(* IEC 61131-3 sources: teller/JD_Teller_LC2_V11/Class/_AlarmX0Para, 1 file *)

(* ---- _AlarmX0Para.st ---- *)
(*!
<Class
	Name               = "_AlarmX0Para"
	Revision           = "0.4"
	RealtimeTask       = "false"
	CyclicTask         = "false"
	BackgroundTask     = "false"
	Sigmatek           = "true"
	OSInterface        = "false"
	HighPriority       = "false"
	Automatic          = "false"
	UpdateMode         = "Prescan"
	SharedCommandTable = "true"
	Objectsize         = "(284,120)">
	<Channels>
		<Server Name="ClassSvr" Visualized="true" Initialize="false" WriteProtected="false" Retentive="false"/>
		<Client Name="Acknow" Required="false" Internal="false"/>
		<Client Name="Config" Required="true" Internal="false" DefValue="0"/>
		<Client Name="Group" Required="false" Internal="false"/>
	</Channels>
	<RevDoku>
		<Owner Company="sigmatek" Author="kolott"/>
		<Dokumentation Revision="0.4" Date="2013-10-30" Author="kolott" Company="sigmatek" Description="sa26144: instances of class _AlarmX0Para will work without instance of class _AlarmXBuffer"/>
		<Dokumentation Revision="0.3" Date="2013-03-19" Author="kolott" Company="sigmatek" Description="innovation: global pointer to _AlarmXBuffer is in use"/>
	</RevDoku>
</Class>
*)
_AlarmX0Para : CLASS
	TYPE
	  yyyy : ^_AlarmXBuffer;
	END_TYPE
  //Servers:
	ClassSvr 	: SvrChCmd_DINT;
  //Clients:
	Config 	: CltCh_DINT;
	Acknow 	: CltCh_DINT;
	Group 	: CltCh_DINT;
  //Variables:
  //Functions:

	FUNCTION _AlarmX0Para
		VAR_OUTPUT
			ret_code 	: ConfStates;
		END_VAR;

	FUNCTION VIRTUAL GLOBAL Init;

	FUNCTION VIRTUAL GLOBAL GetParaID
		VAR_INPUT
			ppara 	: ^UDINT;
		END_VAR
		VAR_OUTPUT
			retcode 	: UDINT;
		END_VAR;

	FUNCTION VIRTUAL GLOBAL GetParaVal
		VAR_INPUT
			ppara 	: ^DINT;
		END_VAR
		VAR_OUTPUT
			retcode 	: UDINT;
		END_VAR;

	FUNCTION GLOBAL QuitAlarm;

	FUNCTION VIRTUAL GLOBAL ClassSvr::Write
		VAR_INPUT
			input (EAX) 	: DINT;
		END_VAR
		VAR_OUTPUT
			result (EAX) 	: DINT;
		END_VAR;
  //Tables:
	FUNCTION @STD
		VAR_OUTPUT
			ret_code	: CONFSTATES;
		END_VAR;
	FUNCTION GLOBAL TAB @CT_;
END_CLASS;

#pragma usingLtd _AlarmXBuffer

#pragma using _AlarmXBuffer

VAR_EXTERNAL
  PV_AlarmBuffer : ^_AlarmXBuffer;
END_VAR

FUNCTION  _AlarmX0Para::_AlarmX0Para
VAR_OUTPUT
	ret_code		: CONFSTATES;
END_VAR

  Acknow         := 0;
  PV_AlarmBuffer :=NIL;
  ret_code       := C_OK;

END_FUNCTION
FUNCTION VIRTUAL GLOBAL _AlarmX0Para::Init
  VAR
    p0    : ^VirtualBase;
    paras : ARRAY[0..MAX_ALARMPARA-1] of UDINT;
    anz   : UDINT;
  END_VAR

  if(_firstscan = 1) then
    _memset(#paras[0], 0, sizeof(paras));
    Config := Config.Read();
    Group  := Group.Read();
    anz    := GetParaID(#paras[0]);

    if(PV_AlarmBuffer = NIL) then
      _LookUpEmbed_C("_AlarmXBuffer1", #PV_AlarmBuffer, #p0);
    end_if;

    if(PV_AlarmBuffer <> NIL) then
      Config$UDINT := PV_AlarmBuffer^.RegisterAlarmXPara(this, Config$UDINT, Group$UDINT, anz, #paras[0]);
    end_if;
  end_if;

END_FUNCTION
FUNCTION GLOBAL _AlarmX0Para::QuitAlarm

  if(Acknow = 0) then
    Acknow := 1;
    if(IsClientConnected(#Acknow) = TRUE) then
      Acknow.Write(Acknow);
    end_if;

    if(PV_AlarmBuffer <> NIL) then
      Config := Config.Read();
      PV_AlarmBuffer^.ActionAlarm(this$UDINT, Config$UDINT, 0, -1, 0, NIL);
    end_if;
  end_if;

END_FUNCTION
FUNCTION VIRTUAL GLOBAL _AlarmX0Para::ClassSvr::Write
VAR_INPUT
	input		: DINT;
END_VAR
VAR_OUTPUT
	result		: DINT;
END_VAR
VAR
  paras : ARRAY[0..MAX_ALARMPARA-1] of DINT;
  anz : udint;
END_VAR

  if(input = 255) then
    QuitAlarm();
  else
    if(ClassSvr <> input) then
      if(PV_AlarmBuffer <> NIL) then
        Acknow   := 0; // prepaire alarm to quit
        ClassSvr := input;
        Group    := Group.Read();
        anz      := GetParaVal(#paras[0]);
        PV_AlarmBuffer^.ActionAlarm(this$UDINT, Config$UDINT, Group$UDINT, ClassSvr, anz, #paras[0]);
      end_if;
    end_if;
  end_if;

  result := 0;

END_FUNCTION
#pragma warning (disable:73)
FUNCTION VIRTUAL GLOBAL _AlarmX0Para::GetParaID
  VAR_INPUT
    ppara		: ^UDINT;
  END_VAR
  VAR_OUTPUT
    retcode		: UDINT;
  END_VAR

  retcode := 0;

END_FUNCTION
FUNCTION VIRTUAL GLOBAL _AlarmX0Para::GetParaVal
VAR_INPUT
	ppara		: ^DINT;
END_VAR
VAR_OUTPUT
	retcode		: UDINT;
END_VAR

  retcode := 0;

END_FUNCTION
#pragma warning (default:73)
